// Mitsubishi GX Works2 project: 0319_인터로크   PLC: Q03UDV

PROGRAM MAIN
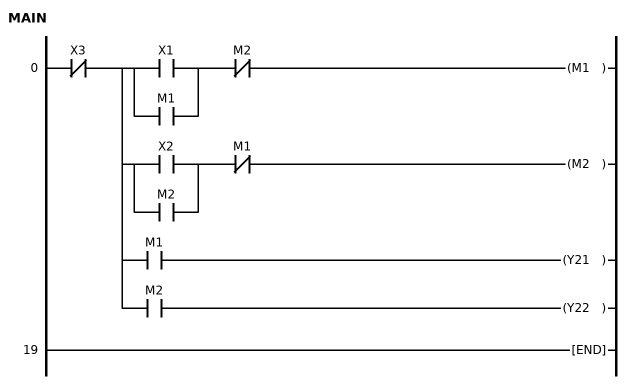
0     LDI     X3
      MPS
      LD      X1
      OR      M1
      ANB
      ANI     M2
      OUT     M1
      MRD
      LD      X2
      OR      M2
      ANB
      ANI     M1
      OUT     M2
      MRD
      AND     M1
      OUT     Y21
      MPP
      AND     M2
      OUT     Y22
19    END
END_PROGRAM
